FUNCTION_BLOCK CylinderHSens (* Composite Function Block Type *)
  (* Standard: 61499-2 *)
  (* Version 0.0, 5/28/2016, Andrei, nxtControl GmbH, template *)
  PACKAGE Main;
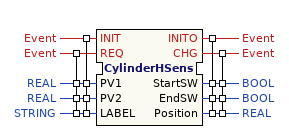
  EVENT_INPUT
    INIT WITH PV1, PV2, LABEL;
    REQ WITH PV1, PV2, LABEL; (* Normal Execution Request *)
  END_EVENT
  EVENT_OUTPUT
    INITO WITH StartSW, EndSW, Position;
    CHG WITH StartSW, EndSW, Position; (* Execution Confirmation *)
  END_EVENT
  VAR_INPUT
    PV1 : REAL; (* Input event qualifier *)
    PV2 : REAL;
    LABEL : STRING;
  END_VAR
  VAR_OUTPUT
    StartSW : BOOL; (* Output event qualifier *)
    EndSW : BOOL;
    Position : REAL;
  END_VAR
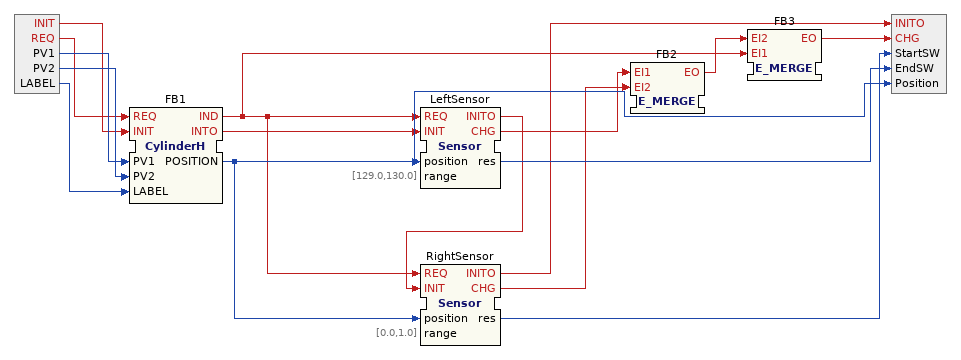
  FBS
    LeftSensor : Sensor(range := [129.0,130.0]);
    RightSensor : Sensor(range := [0.0,1.0]);
    FB1 : CylinderH;
    FB2 : E_MERGE;
    FB3 : E_MERGE;
  END_FBS
  EVENT_CONNECTIONS
    REQ TO FB1.REQ;
    FB1.IND TO RightSensor.REQ;
    FB1.IND TO LeftSensor.REQ;
    FB3.EO TO CHG;
    INIT TO FB1.INIT;
    RightSensor.INITO TO INITO;
    LeftSensor.INITO TO RightSensor.INIT;
    FB1.INTO TO LeftSensor.INIT;
    FB2.EO TO FB3.EI2;
    LeftSensor.CHG TO FB2.EI1;
    RightSensor.CHG TO FB2.EI2;
    FB1.IND TO FB3.EI1;
  END_CONNECTIONS
  DATA_CONNECTIONS
    PV1 TO FB1.PV1;
    PV2 TO FB1.PV2;
    LABEL TO FB1.LABEL;
    FB1.POSITION TO LeftSensor.position;
    FB1.POSITION TO RightSensor.position;
    RightSensor.res TO StartSW;
    LeftSensor.res TO EndSW;
    FB1.POSITION TO Position;
  END_CONNECTIONS
END_FUNCTION_BLOCK
